                IF (configuration.power.syncMotionSimulation = TRUE) THEN
                   (* SynchroniziedMotionSimulation is set*)
                    IF (tempEnableAxis = FALSE) AND (statEnableAxisOld = TRUE) THEN
                       (* Falling edge at enableAxis --> set simulation*)
                        statSyncMotionSimulationState := AXIS_STATE_SET_SIM;
                        statEnableAxis                := TRUE;
                        tempStateChangeActive         := TRUE;
                    ELSE
                       (* FALSE or rising edge at input enableAxis*)
                        statEnableAxis := tempEnableAxis;
                    END_IF;

                ELSE
                   (* SynchroniziedMotionSimulation not set*)
                   (* MC_POWER is only controlled by enableAxis input*)
                    statEnableAxis := tempEnableAxis;
                END_IF;

            AXIS_STATE_SET_SIM:
				(*
                (* Set the axis in simulation*)
                (*----------------------------------------------------------*)
                (* Enable SynchronizedMotionSimulation*)
				*)
                instSyncMotionSimulation(Slave := axis,
                                         Enable := TRUE);
				(*
                (*----------------------------------------------------------*)
				*)
				
                IF (instSyncMotionSimulation.InSimulation = TRUE) THEN
                    statEnableAxis := FALSE;
                   (* Axis in Simulation - Change state*)
                    statSyncMotionSimulationState := AXIS_DISABLE;

                ELSIF (instSyncMotionSimulation.Error = TRUE) THEN
                   (* Error occurred - Disable Axis immediately*)
                    statEnableAxis                := FALSE;
                    statSyncMotionSimulationState := AXIS_STATE_RESET_SIM;

                ELSE
                    ;(* Wait for Axis is in simulation*)
                END_IF;

            AXIS_DISABLE:

                (* Disable axis*)
                (*----------------------------------------------------------*)
                (* Enable SynchronizedMotionSimulation*)

                instSyncMotionSimulation(Slave := axis,
                                         Enable := TRUE);

                (*----------------------------------------------------------*)


                IF (instPower.Error = TRUE) THEN
                    statSyncMotionSimulationState := AXIS_STATE_RESET_SIM;
                ELSIF (instPower.Status = FALSE) THEN
                   (* Axis disabled*)
                    statSyncMotionSimulationState := AXIS_STATE_IN_SIM;
                ELSE
                    ;(* Wait for Axis is disabled*)
                END_IF;

            AXIS_STATE_IN_SIM:

                (* Axis is in simulation*)
                (*----------------------------------------------------------*)
                (* Enable SynchronizedMotionSimulation*)

                instSyncMotionSimulation(Slave := axis,
                                         Enable := TRUE);

                (*----------------------------------------------------------*)

				
                IF (tempEnableAxis = TRUE) AND (statEnableAxisOld = FALSE) THEN
                   (* Rising edge at enableAxis --> reset simulation*)
                    statSyncMotionSimulationState := AXIS_ENABLE;
                    statEnableAxis                := TRUE;
                    tempStateChangeActive         := TRUE;
                ELSIF (configuration.power.syncMotionSimulation = FALSE) THEN
                   (* End of synchronizedMotionSimulation by configuration without starting Axis*)
                    statSyncMotionSimulationState := AXIS_STATE_RESET_SIM;
                    tempStateChangeActive         := TRUE;

                ELSE
                    ;(* Wait for rising egde at enableAxis*)
                END_IF;

            AXIS_ENABLE:

                (* Enable Axis*)
                (*----------------------------------------------------------*)
                (* Enable SynchronizedMotionSimulation while axis is enabling*)
				
                instSyncMotionSimulation(Slave := axis,
                                         Enable := TRUE);


                (*----------------------------------------------------------*)
                (* Read Statusword only when not already read out*)

                IF (tempStatusWord = 16#0)
                    THEN

                    (*tempStatusWord :=  axis.StatusWord;*)
                    tempStatusWord := axis.NcToPlc.StateDWord;

                END_IF;

                IF (tempEnableAxis = FALSE) AND (statEnableAxisOld = TRUE) THEN
                    statSyncMotionSimulationState := AXIS_STATE_RESET_SIM;
                    statEnableAxis                := FALSE;

                ELSIF (tempStatusWord.0 = TRUE) OR (instPower.Error = TRUE)
               (* Reset simulation if axis is enabled or MC_POWER.STATUS = FALSE (Axis Error)*)
                    THEN
                   (* FALSE on enable input*)
                    statSyncMotionSimulationState := AXIS_STATE_RESET_SIM;
                    tempStateChangeActive         := TRUE;

                ELSE
                    ;(* Wait for Axis is Enabled*)
                END_IF;

            AXIS_STATE_RESET_SIM:

                (* Reset the axis simulation*)
                (*----------------------------------------------------------*)
                (*Enable SynchronizedMotionSimulation*)
				

                instSyncMotionSimulation(Slave := axis,
                                         Enable := FALSE);

                (*----------------------------------------------------------*)

				
                IF (instSyncMotionSimulation.InSimulation = FALSE) AND
                    (instSyncMotionSimulation.Busy = FALSE)
                    THEN
                   (* Axis simulation is disabled*)
                    statSyncMotionSimulationState := AXIS_NOT_IN_SIM;

                ELSE
                    ;(* Wait for axis simulation is disabled*)
                END_IF;

                IF (tempEnableAxis = FALSE) AND (statEnableAxisOld = TRUE) THEN
                    statEnableAxis := FALSE;
                END_IF;

        ELSE
           (* Errorhandling*)
            statStatus                          := ERR_UNDEFINED_MOTION_SIMULATION_STATE;
            statErrorUserCleared                := TRUE;
            diagnostics.subfunctionStatus       := 0;
            diagnostics.basicMotionState        := statBasicMotionState;
            diagnostics.superimposedMotionState := statSupImpMotionState;
           (* Set error state*)
            statFBState := FB_ERROR;
        END_CASE;
    UNTIL (tempStateChangeActive = FALSE)
    END_REPEAT;

   (* Evaluation of MC_Command*)
    IF (instSyncMotionSimulation.Error = TRUE) AND (statSynchronizedMotionErrorOld = FALSE) THEN
       (* Errorhandling - Set error only at rising edge*)
        statErrorAutoCleared                := TRUE;
        statStatus                          := ERR_MC_SYNCHRONIZEDMOTIONSIMULATION;
        diagnostics.basicMotionState        := statBasicMotionState;
        diagnostics.superimposedMotionState := statSupImpMotionState;
        diagnostics.subfunctionStatus       := instSyncMotionSimulation.ErrorId;

    ELSIF (instSyncMotionSimulation.Error = FALSE) AND (statStatus = ERR_MC_SYNCHRONIZEDMOTIONSIMULATION)
        THEN
       (* Reset error if error gone at respective Status*)
        statErrorAutoCleared := FALSE;
        statStatus           := STATUS_SUBSEQUENT_CALL;
    ELSE
        ;
    END_IF;

    statSynchronizedMotionErrorOld := instSyncMotionSimulation.Error;
    tempEnableAxis                 := statEnableAxis;
    {END_REGION}

   (* Enable and disable axis*)
    {REGION "POWER"}
   (* Call MC_POWER*)
    instPower(Axis := axis,
              	Enable := tempEnableAxis,
              	Enable_Positive := TRUE,
            	Enable_Negative := TRUE,
    		(*StartMode :=  configuration.power.startMode,
	         StopMode :=  configuration.power.stopMode*) );

   (* Set and Reset of Error*)
    IF (instPower.Error = TRUE) AND
        ((statStatus = STATUS_SUBSEQUENT_CALL) OR (statPowerErrorOld = FALSE))
        THEN
       (* Error is set at rising edge of MC_POWER.Error*)
       (* Errorhandling*)
        statStatus                              := ERR_MC_POWER;
        statErrorAutoCleared                    := TRUE;
        statDiagnostics.basicMotionState        := statBasicMotionState;
        statDiagnostics.superimposedMotionState := statSupImpMotionState;
        statDiagnostics.subfunctionStatus       := instPower.ErrorId;
        diagnostics                             := statDiagnostics;

    ELSIF (statStatus = ERR_MC_POWER) AND (instPower.Error = FALSE)
        THEN
       (* Reset Error*)
        statStatus           := STATUS_SUBSEQUENT_CALL;
        statErrorAutoCleared := FALSE;

    ELSIF (tempEnableAxis = TRUE) AND (statEnableAxisOld = FALSE) THEN
       (* Reset Error*)
        statStatus           := STATUS_SUBSEQUENT_CALL;
        statErrorAutoCleared := FALSE;
        diagnostics          := statEmptyDiagnostics;
        statDiagnostics      := statEmptyDiagnostics;

    ELSE
        ;(* Do nothing*)
    END_IF;
    {END_REGION}
    {END_REGION}
END_IF;

{END_REGION}


(*----------------------------------------------------------------------------------------------*)
(*FB Statemachine *)
(*----------------------------------------------------------------------------------------------*)


{REGION "FB_STATEMACHINE"}
CASE statFBState OF
    AXIS_MOTION:
       (* Check command inputs*)
        IF (statExtendedCommand = CMD_NO_SELECTION) AND (statBasicCommand = CMD_NO_SELECTION) AND (statSupImpCommand = CMD_NO_SELECTION)
            THEN
           (* Command is reset*)
            IF (instPower.Error = TRUE) THEN
               (* Errorhandling*)
                statStatus           := ERR_MC_POWER;
                statErrorAutoCleared := TRUE;
                diagnostics          := statDiagnostics;
            ELSIF (instSyncMotionSimulation.Error = TRUE) THEN
                ;(* Do nothing*)

            ELSIF (instTorqueLimiting.Error = TRUE) THEN
                ;(* Do nothing. V1.00.03 dont reset IF torque limiting  error is pending *)

            ELSE
               (* Reset Error only if no Error at MC_POWER is present*)
                statStatus           := STATUS_SUBSEQUENT_CALL;
                statErrorAutoCleared := FALSE;
            END_IF;

        ELSIF (statExtendedCommand = statExtendedCommandOld) AND
            (statBasicCommand = statBasicCommandOld) AND
            (statSupImpCommand = statSupImpCommandOld)
            THEN
            ;(* No change at command - do nothing*)

        ELSE
           (* Command changed*)
            tempNewExtendedCmd    := NO_SELECTION;
            tempNewBasicMotionCmd := NO_SELECTION;
            tempNewSupImpCmd      := NO_SELECTION;
            tempErrorInCmd        := FALSE;

            {REGION "CHECK BASIC_MOTION_CMD"}
           (* Check basic motion command*)
            IF (statBasicCommand = statBasicCommandOld) THEN
                ;(* Do nothing*)
            ELSE
               (* Evaluate rising edges for basic motion command word - all rising edges of basic command word saved in tempRisingBasicCmd*)
                tempRisingCmd     := ((statBasicCommand XOR statBasicCommandOld) AND statBasicCommand);
                tempCountRisEdges := 0;(* Initialize counter for rising edges*)
               (* Count rising edges in tempRisingBasicCmd*)
                FOR tempIndex := BITPOSITION_BASIC_MOTION_CMD TO BIT_POS_LAST DO
                    tempDword := SHR(tempRisingCmd, INT_TO_USINT(tempIndex));
                   (* Check for rising edge*)
                    IF (tempDword.0 = TRUE) THEN
                        tempCountRisEdges := tempCountRisEdges + 1;(* Increment at rising edge*)
                    END_IF;
                END_FOR;

                IF (tempRisingCmd.2 = TRUE) OR (tempRisingCmd.3 = TRUE) THEN
                    tempCountRisEdges := tempCountRisEdges + 1;(* jogForward AND/OR jogBackward is standing for 1 Command/rising edge*)
                END_IF;

               (* Check Basic motion command*)
                IF (tempCountRisEdges = 1) OR
                    (tempRisingCmd.0 = TRUE)(* fastStop selected*)
                    OR
                    (tempRisingCmd.1 = TRUE)(* Stop selected*)
                    THEN
                   (* Valid basic motion command selected*)
                    IF (tempRisingCmd.0 = TRUE)
                        THEN
                       (* FastStop selected*)
                        statFBState           := AXIS_FAST_STOPPING;
                        tempNewBasicMotionCmd := FAST_STOP_SELECTED;
                        tempStopCmdSelected   := TRUE;
                    ELSIF (tempRisingCmd.1 = TRUE)
                        THEN
                       (* Stop selected*)
                        tempNewBasicMotionCmd := STOP_SELECTED;
                        tempStopCmdSelected   := TRUE;
                    ELSE
                       (* Valid basic command priority 3 selected*)
                       (* Set basic motion state*)
                        tempNewBasicMotionCmd := DWORD_TO_DINT(tempRisingCmd);
                    END_IF;

                ELSIF (tempCountRisEdges > 1) THEN
                   (* Errorhandling - Invalid command *)
                    statStatus     := ERR_INVALID_BASIC_MOTION_CMD;
                    tempErrorInCmd := TRUE;

                ELSE
                    ;(* Falling edge detection*)
                END_IF;
            END_IF;

            {END_REGION}
            {REGION "CHECK_SUP_IMP_CMD"}
           (* Check superimposed motion command*)
            IF (statSupImpCommand = statSupImpCommandOld) THEN
                ;(* Do nothing*)
            ELSE
               (* Superimposed motion command selected *) 
                IF (tempErrorInCmd = FALSE) AND(* No Stop command selected in current cycle*)
                    (tempStopCmdSelected = FALSE)
                    THEN
                    tempRisingCmd     := ((statSupImpCommand XOR statSupImpCommandOld) AND statSupImpCommand);
                    tempCountRisEdges := 0;(* Initialize counter for rising edges*)
                   (* Count rising edges in tempRisingSupImpCmd*)
                    FOR tempIndex := BITPOSITION_SUPERIMPOSED_MOTION_CMD TO BIT_POS_LAST DO
                        tempDword := SHR(tempRisingCmd, INT_TO_USINT(tempIndex));
                       (* Check for rising edge*)
                        IF (tempDword.0 = TRUE) THEN
                            tempCountRisEdges := tempCountRisEdges + 1;
                        END_IF;
                    END_FOR;

                    IF (tempCountRisEdges = 1) THEN
                       (* Valid superimposed motion command*)
                        tempNewSupImpCmd := DWORD_TO_DINT(tempRisingCmd);

                    ELSIF (tempCountRisEdges > 1) THEN
                       (* Invalid Superimposed motion command*)
                        statStatus     := ERR_INVALID_SUPERIMPOSED_MOTION_CMD;
                        tempErrorInCmd := TRUE;

                    ELSE
                        ;(* Falling edge detection*)
                    END_IF;

                ELSE
                    ;(* Stop or Faststop command selected OR error in BasicCommand*)
                END_IF;
            END_IF;

            {END_REGION}
            {REGION "CHECK_EXT_CMD"}
           (* Check extended command (reset, homing, torquelimiting)*)
            IF (statExtendedCommand = statExtendedCommandOld) THEN
                ;(* Do nothing*)
            ELSE
               (* Extended command selected*)
                IF (tempErrorInCmd = FALSE)
                    THEN
                    tempRisingCmd := ((statExtendedCommand XOR statExtendedCommandOld) AND statExtendedCommand);
                   (* Rising edge on torquelimiting command*)
                    IF (tempRisingCmd.1 = TRUE)
                        THEN
                        tempNewExtendedCmd.1 := TRUE;
                       (* Rising Edge at Homing on Fixed Stop and Torquelimiting*)
                        IF (tempNewBasicMotionCmd.10 = TRUE) AND (configuration.homing.extendedMode = 0) THEN
                            ;(* Errorhandling*)
                            statStatus           := ERR_INVALID_EXTENDED_CMD;
                            tempErrorInCmd       := TRUE;
                            tempNewExtendedCmd.1 := FALSE;

                           (* Check if torquelimiting is not for use in homing on fixed stop function*)
                        ELSIF (statTorqueLimitingState = TORQUE_LIMTING_SELECTED)
                       (* OR ( statTorqueLimitingState =  AUTOMATIC_MODE_CHANGE) V1.00.03 Not required anymore*)
                            THEN
                            ;(* Torquelimiting already busy no need of restart*)
                           (* tempNewExtendedCmd.1 := FALSE; // V1.0.4 Initialize Diagnostics at rising edge of torquelimiting*)

                        ELSIF (statTorqueLimitingState = FIXED_STOP_DETECTION_ACTIVE)
                            THEN
                            ;(* Torquelimiting rejected because MC_Torquelimiting is used during homing on fixed stop functionality*)
                            statStatus           := ERR_TORQUE_LIMITING_NOT_ALLOWED;
                            tempErrorInCmd       := TRUE;
                            tempNewExtendedCmd.1 := FALSE;

                        ELSE
                            ;(* Start torquelimiting functionality*)
                        END_IF;
                    END_IF;

                   (* Rising edge on passive homing command*)
                    IF (tempRisingCmd.2 = TRUE)
                        THEN
                        tempNewExtendedCmd.2 := TRUE;
                        IF (statBasicMotionState = ACTIVE_HOMING_SELECTED) AND
                            (statActiveHomingState = HOMING_ON_FIXED_STOP) AND
                            (statExeOfBasicMotion = CMD_BUSY)
                            THEN
                           (* Passive Homing selected at homing on fixed stop *)
                            statStatus           := ERR_HOMING_MODE_NOT_ALLOWED;
                            tempErrorInCmd       := TRUE;
                            tempNewExtendedCmd.2 := FALSE;
                        ELSE
                            ;(* No error occurred*)
                        END_IF;
                    END_IF;
                ELSE
                    ;(* Error in basic motion command or superimposed motion command *)
                END_IF;
            END_IF;

            {END_REGION}
           (* Enable commands*)
            IF (tempErrorInCmd = TRUE) AND (tempStopCmdSelected = FALSE)
                THEN
               (* Error in current command - No Execution*)
                statErrorAutoCleared          := TRUE;
                diagnostics.subfunctionStatus := 0;
               (* Write diagnostics*)
                statDiagnostics.basicMotionState        := statBasicMotionState;
                statDiagnostics.superimposedMotionState := statSupImpMotionState;
                statResetIncJog                         := TRUE;
               (* Set next state*)
                statFBState := AXIS_STOP_ON_ERROR_SELECTION;
            ELSE
               (* No Error in command occurred*)
                IF (
                    (tempNewExtendedCmd <> NO_SELECTION) OR (tempNewBasicMotionCmd <> NO_SELECTION) OR (tempNewSupImpCmd <> NO_SELECTION)
                    ) OR
                    (tempStopCmdSelected = TRUE)
                    THEN
                    {REGION "ENABLE_BASIC_MOTION_CMD"}
                   (* New valid command selected*)
                   (* Basic motion commands*)
                    IF (tempNewBasicMotionCmd <> NO_SELECTION) THEN
                       (* Reset of waiting Gearin / camIn command*)
                        IF (configuration.generalSettings.abortWaitingSyncCmd = TRUE) AND
                            (((statBasicMotionState = GEAR_IN_ABSOLUTE_SELECTED) AND (statExeOfBasicMotion = CMD_BUSY))(* GearInAbsolute waiting*)
                            OR
                            ((statBasicMotionState = CAM_IN_SELECTED) AND (statExeOfBasicMotion = CMD_BUSY)))(* CamIn waiting*)
                            THEN
                            statMainSelectionState := RESET_GEARING;(* Reset waiting absolute gearing / camIn command *)
                            instGearIn(Master := master,
                                       Slave := axis,
                                       Execute := FALSE);
                        ELSE
                            statMainSelectionState := CALL_BASIC_MOTION;
                        END_IF;

                        statFirstCycleBasicMotion := TRUE;
                       (* Evaluate if Jog command is set*)
                        IF (tempNewBasicMotionCmd.2 = TRUE) OR (tempNewBasicMotionCmd.3 = TRUE)
                            THEN
                            statExeOfBasicMotion := CMD_BUSY;
                           (* Select Jogmode*)
                            IF ((statBasicCommand.2 = FALSE) AND (tempNewBasicMotionCmd.3 = TRUE)
                                ) OR(* Rising edge at JogBackward and JogForward = FALSE*)
                                ((statBasicCommand.3 = FALSE) AND (tempNewBasicMotionCmd.2 = TRUE)
                                ) OR(* Only rising edge at JogForward and Jogbackward = FALSE*)
                                ((tempNewBasicMotionCmd.2 = TRUE) AND (tempNewBasicMotionCmd.3 = TRUE)
                                )(* Rising edge at FW and BW*)
                                THEN
                               (* One Input direction = False, other is rising edge, or both rising edge --> Start jog*)
                                IF (statJogMode <> configuration.jog.mode) THEN
                                    statResetIncJog := TRUE;
                                END_IF;

                                statJogMode := configuration.jog.mode;
                            ELSE
                                ;(* Rising edge at one input, the other is already TRUE - Dont Change Jogmode*)
                                IF ((statBasicMotionState = JOG_BACKWARD_SELECTED) OR (statBasicMotionState = JOG_FORWARD_SELECTED)) AND
                                    (statJogMode <> JOG_MODE_CONTINUOUS)
                                    THEN
                                    statFirstCycleBasicMotion := FALSE;
                                END_IF;
                            END_IF;

                        ELSE
                            ;(* Reset jog increment if other command than jog selected*)
                            statResetIncJog := TRUE;
                        END_IF;

                       (* Set new basic motion state*)
                        statBasicMotionState := tempNewBasicMotionCmd;
                    END_IF;

                    {END_REGION}
                    {REGION "ENABLE_SUP_IMP_CMD"}
                   (* Superimposed motion commands*)
                    IF (tempNewSupImpCmd <> NO_SELECTION) THEN
                        statSupImpMotionState      := tempNewSupImpCmd;
                        statFirstCycleSupImpMotion := TRUE;
                        statResetIncJog            := TRUE;
                    END_IF;

                    {END_REGION}
                   (* Extended commands*)
                    {REGION "ENABLE_EXT_CMD"}
                    IF (tempNewExtendedCmd <> NO_SELECTION) THEN
                        IF (tempNewExtendedCmd.1 = TRUE) THEN
                           (* Rising edge on torquelimiting command*)
                            IF (statTorqueLimitingState = NO_TORQUE_LIMITING_ACTIVE)
                                THEN
                               (* No torquelimiting active --> Enable torquelimiting*)
                                statTorqueLimitingState := TORQUE_LIMTING_SELECTED;
                            ELSE
                                ;(* Torquelimiting already active*)
                               (* statTorqueLimitingState :=  AUTOMATIC_MODE_CHANGE; V1.00.03 Not required anymore *)
                            END_IF;
                        END_IF;

                       (* Homing command*)
                        IF (tempNewExtendedCmd.2 = TRUE) THEN
                            statPassiveHomingState := configuration.homing.extendedMode;
                            statFirstCycleHoming   := TRUE;
                            statResetIncJog        := TRUE;
                        END_IF;
                    END_IF;

                    {END_REGION}
                   (* Reset error*)
                    statStatus           := STATUS_SUBSEQUENT_CALL;
                    statErrorAutoCleared := FALSE;
                    diagnostics          := statEmptyDiagnostics;
                    statDiagnostics      := statEmptyDiagnostics;

                ELSE
                    ;(* No rising edge at commands*)
                END_IF;
            END_IF;
        END_IF;

    AXIS_FAST_STOPPING:
        IF (configuration.fastStop.replaceStopPossible = FALSE) THEN
            ;(* Fast stop command can not be interrupted by another command*)
           (* State change is executed in FastStop implementation if command finished *)
        ELSE
            statFBState := AXIS_MOTION;
        END_IF;

    AXIS_STOP_ON_ERROR_SELECTION,
        AXIS_STOP_ON_ERROR_EXECUTION:
        ;    (* Wait for stopping axis if StopOnError is configured*)
    FB_ERROR:(* Error state*)
        ;    (* Do nothing, status already set*)

ELSE
   (* Errorhandling*)
    statStatus                          := ERR_UNDEFINED_FB_STATE;
    statErrorUserCleared                := TRUE;
    diagnostics.subfunctionStatus       := 0;
    diagnostics.basicMotionState        := statBasicMotionState;
    diagnostics.superimposedMotionState := statSupImpMotionState;
   (* Set error state*)
    statFBState := FB_ERROR;
END_CASE;

{END_REGION}


(*----------------------------------------------------------------------------------------------*)
(*Execution of reset functionality*)
(*----------------------------------------------------------------------------------------------*)


{REGION "EXECUTION_OF_RESET_COMMAND"}
(* Firstcycle of command*)

IF (statExtendedCommand.0 = TRUE) AND (statExtendedCommandOld.0 = FALSE) THEN
    statFirstCycleReset := TRUE;
   (* Reset MC_RESET command*)
    instReset(Axis := axis,
              Execute := FALSE);

    statFirstCycleResetError := FALSE;
    statResetState           := CMD_BUSY;
END_IF;

CASE statResetState OF
    CMD_IDLE:
        ;(* Do nothing*)

    CMD_BUSY:
       (* Call MC_Command*)
        instReset(Axis := axis,
                  Execute := statExtendedCommand.0,
        (*Restart :=  configuration.generalSettings.resetWithRestart*) );

       (* Evaluate MC_Command*)
        IF (instReset.Error = TRUE) THEN
           (* Errorhandling*)
            IF (statFirstCycleResetError = FALSE) THEN
                statErrorAutoCleared                := TRUE;
                diagnostics.status                  := ERR_MC_RESET;
                statStatus                          := ERR_MC_RESET;
                diagnostics.basicMotionState        := statBasicMotionState;
                diagnostics.superimposedMotionState := statSupImpMotionState;
                diagnostics.subfunctionStatus       := instReset.ErrorId;
                statFirstCycleResetError            := TRUE;
               (* Set next state*)
                statResetState := CMD_IDLE;
                IF (statFBState = AXIS_MOTION) THEN
                   (* Set TO_STOP_ON_ERROR State only if the current state is TO_MOTION*)
                    statFBState := AXIS_STOP_ON_ERROR_SELECTION;
                END_IF;
            END_IF;

        ELSIF (instReset.Busy = FALSE) THEN
           (* Set next state*)
            statResetState := CMD_IDLE;
        ELSE
            ;(* Command selected*)
        END_IF;

ELSE
   (* Errorhandling  *)  
    statStatus                              := ERR_UNDEFINED_RESET_STATE;
    statErrorUserCleared                    := TRUE;
    diagnostics                             := statDiagnostics;
    diagnostics.subfunctionStatus           := 0;
    statDiagnostics.basicMotionState        := statBasicMotionState;
    statDiagnostics.superimposedMotionState := statSupImpMotionState;
END_CASE;

{END_REGION}


(*----------------------------------------------------------------------------------------------*)
(* Execution of functionalities of basic coordinate system*)
(*----------------------------------------------------------------------------------------------*)


{REGION "EXECUTION_OF_BASIC_MOTION_COMMANDS"}
(*Statemachine for basic motion commands*)

(*Write diagnostics*)
statDiagnostics.basicMotionState        := statBasicMotionState;
statDiagnostics.superimposedMotionState := statSupImpMotionState;
REPEAT
    tempStateChangeActive := FALSE;
   (* Statemachine for main selection state*)
    CASE statMainSelectionState OF
        CALL_BASIC_MOTION:
            CASE statBasicMotionState OF
                NO_SELECTION:
                    ;(* No execution*)

                FAST_STOP_SELECTED:
                    ;(* Implementation at end of code*)

                STOP_SELECTED:
                   (* No additional features*)
                    {REGION "STOP_SELECTED"}
                   (* Firstcycle of command*)
                    IF (statFirstCycleBasicMotion = TRUE) THEN
                       (* Reset HALT command*)
                        instHalt(Axis := axis,
                                 Execute := FALSE);
                    END_IF;

                   (* Call MC_Command*)
                    instHalt(Axis := axis,
                             Execute := statBasicCommand.1 OR statFirstCycleBasicMotion,
                             Deceleration := configuration.stop.deceleration,
                             (*AbortAcceleration :=  configuration.stop.abortAcceleration,*)
                             Jerk := configuration.stop.jerk);

                   (* Evaluate MC_Command*)
                    IF (instHalt.Busy = FALSE) AND
                        (instHalt.Error = FALSE) AND
                        (instHalt.Done = FALSE) AND
                        (instHalt.CommandAborted = FALSE)
                        THEN
                       (* Return to NO_SELECTION if command finished*)
                        statBasicMotionState := NO_SELECTION;

                    ELSIF (instHalt.Error = TRUE)
                        THEN
                       (* Errorhandling*)
                        statStatus                    := ERR_MC_HALT;
                        statErrorAutoCleared          := TRUE;
                        diagnostics                   := statDiagnostics;
                        diagnostics.subfunctionStatus := instHalt.ErrorId;
                       (* Set next state*)
                        statFBState          := AXIS_STOP_ON_ERROR_SELECTION;
                        statBasicMotionState := NO_SELECTION;
                    ELSE
                        ;(* Command selected*)
                    END_IF;

                   (* Write MC_Command outputs to internal variable*)
                    statExeOfBasicMotion   := 16#0;
                    statExeOfBasicMotion.0 := instHalt.Busy;
                    statExeOfBasicMotion.1 := instHalt.Done;
                    statExeOfBasicMotion.2 := instHalt.CommandAborted;
                    statExeOfBasicMotion.3 := instHalt.Error;
                {END_REGION}

                JOG_FORWARD_SELECTED, JOG_BACKWARD_SELECTED, JOG_FW_AND_BW_SELECTED:
                   (* Additional features (applicative): Jog mode incremental*)
                    {REGION "JOG_SELECTED"}
                    CASE statJogMode OF
                        JOG_MODE_CONTINUOUS:
                            {REGION "JOG_MODE_CONTINUOUS"}
                           (* No additional feature*)
                           (* Firstcycle of command*)
                            IF (statFirstCycleBasicMotion = TRUE) THEN
                               (* No of dynmics into static variables because changes are accepted by MC_JOG immetiately (enable)*)
                                instMoveJog(Axis := axis,
                                            JogForward := FALSE,
                                            JogBackwards := FALSE);
                            END_IF;

                           (* Call MC_Command*)
                            instMoveJog(Axis := axis,
                                        JogForward := statBasicCommand.2,
                                        JogBackwards := statBasicCommand.3,
                                        Velocity := configuration.jog.velocity,
                                        Acceleration := configuration.jog.acceleration,
                                        Deceleration := configuration.jog.deceleration,
                                        (*PositionControlled :=  configuration.jog.positionControlled,*)
				Mode := 2,
                                        Jerk := configuration.jog.jerk);

                           (* Evaluate MC_Command*)
                            IF (instMoveJog.Busy = FALSE) AND
                                (instMoveJog.Error = FALSE) AND
                                (instMoveJog.CommandAborted = FALSE) (*AND
	                      ( instMoveJog.InVelocity = FALSE)*)
                                THEN
                               (* Return to NO_SELECTION if command finished*)
                                statBasicMotionState := NO_SELECTION;

                            ELSIF (instMoveJog.Error = TRUE)
                                THEN
                               (* Errorhandling*)
                                statStatus                    := ERR_MC_MOVEJOG;
                                statErrorAutoCleared          := TRUE;
                                diagnostics                   := statDiagnostics;
                                diagnostics.subfunctionStatus := instMoveJog.ErrorId;
                               (* Set next state*)
                                statBasicMotionState := NO_SELECTION;
                                statFBState          := AXIS_STOP_ON_ERROR_SELECTION;

                            ELSE
                                ;(* Command selected*)
                            END_IF;

                           (* Write MC_Command outputs to internal variable*)
                            statExeOfBasicMotion   := 16#0;
                            statExeOfBasicMotion.0 := instMoveJog.Busy;
                            statExeOfBasicMotion.2 := instMoveJog.CommandAborted;
                            statExeOfBasicMotion.3 := instMoveJog.Error;
                            (*statExeOfBasicMotion.4 := instAxisStatus.stAxisStatus.ConstantVelocity; (*####*)*)
				  statExeOfBasicMotion.4 := axis.Status.ConstantVelocity;
                        {END_REGION}

                        JOG_MODE_CONTINUE_INCREMENT, JOG_MODE_NEW_INCREMENT:
                            {REGION "JOG_MODE_INCREMENTAL"}
                           (* This case is additional feature (MC_MOVERELATIVE and MC_HALT internal used)*)
                            CASE statExeOfBasicMotion OF
                                CMD_BUSY:
                                   (* Firstcycle of command*)
                                    IF (statFirstCycleBasicMotion = TRUE) THEN(*New rising edge at JogForward or JogBackard*)
                                       (* Check for only one Jog direction selected (Forward OR Backward)*)
                                        IF (statBasicCommand.2 XOR statBasicCommand.3)(* Only one direction selected*)
                                            THEN
                                           (* Reset MOVERELATIVE command*)
                                            instMoveRelative(Axis := axis,
                                                             Execute := FALSE);

                                           (* Reset HALT command*)
                                            instHalt(Axis := axis,
                                                     Execute := FALSE);

                                           (* Set new Increment if direction changed neccesary*)
                                            IF (statResetIncJog = FALSE) THEN
                                                IF ((statIncJogDirectionOld = FORWARD_DIR) AND (statBasicCommand.2 = TRUE)) OR
                                                    ((statIncJogDirectionOld = BACKWARD_DIR) AND (statBasicCommand.3 = TRUE))
                                                    THEN
                                                    ;(* Direction of last jog process same as current --> continue Jog*)
                                                ELSE
                                                    statResetIncJog := TRUE;
                                                END_IF;
                                            END_IF;

                                           (* Determine distance for positioning command (relative)*)
                                            IF (configuration.jog.mode = JOG_MODE_NEW_INCREMENT)(* In this mode a new increment is always set*)
                                                OR
                                                ((configuration.jog.mode = JOG_MODE_CONTINUE_INCREMENT) AND (statResetIncJog = TRUE))
                                                THEN
                                                statResetIncJog := FALSE;
                                               (* New increment*)
                                                (*statIncJogStartPosition :=  axis.Position;*)              (* Targetposition for increment*)
                                                statIncJogStartPosition := axis.NcToPlc.ActPos;             (* Targetposition for increment*)
                                                statIncrement           := ABS(configuration.jog.increment);(* absolut Distance for increment*)
                                                IF (statBasicCommand.2 = TRUE) THEN
                                                   (* JogForward selected*)
                                                    statPosition           := ABS(configuration.jog.increment);
                                                    statIncrement          := statPosition;
                                                    statIncJogDirectionOld := FORWARD_DIR;
                                                ELSIF (statBasicCommand.3 = TRUE) THEN
                                                   (* JogBackward selected*)
                                                    statPosition           := -ABS(configuration.jog.increment);
                                                    statIncrement          := statPosition;
                                                    statIncJogDirectionOld := BACKWARD_DIR;
                                                ELSE
                                                   (* Normal not possible to reach ELSE-branch*)
                                                    statIncJogDirectionOld := 0;
                                                END_IF;

                                            ELSE
                                               (* Check for modulo axis*)
                                                (*IF ( axis.Modulo.Enable = FALSE) THEN*)
                                                IF (tempFalse = TRUE) THEN
                                                   (* No Modulo enabled*)
                                                   (* Continue increment*)

                                                    statPosition := (statIncJogStartPosition + statIncrement) - axis.NcToPlc.ActPos;
                                                   (* Distance   :=            setpoint                         - actualvalue*)
                                                ELSE
                                                   (* Modulo enabled*)
                                                    statPosition := statIncJogDistance;
                                                END_IF;

                                            END_IF;

                                            statIncJogSubState := INC_JOG_START;

                                           (* Store Dynamics*)
                                            statVelocity     := ABS(configuration.jog.velocity);
                                            statAcceleration := configuration.jog.acceleration;
                                            statDeceleration := configuration.jog.deceleration;
                                            statJerk         := configuration.jog.jerk;

                                        ELSE
                                           (* Errorhandling - Invalid direction (forward and backward selected)*)
                                            statStatus                    := ERR_INVALID_JOG_DIR;
                                            statErrorAutoCleared          := TRUE;
                                            diagnostics.subfunctionStatus := 0;
                                            diagnostics.basicMotionState  := statBasicMotionState;
                                           (* Set next state*)
                                            statFBState          := AXIS_STOP_ON_ERROR_SELECTION;
                                            statBasicMotionState := NO_SELECTION;
                                            statExeOfBasicMotion := CMD_ERROR;
                                            statIncJogSubState   := INC_JOG_IDLE;
                                        END_IF;

                                    ELSIF ((statBasicCommand.2 = FALSE) AND (statBasicCommand.3 = FALSE))(* No jog input selected --> Stop moving*)
                                        AND
                                        (statIncJogSubState <> INC_JOG_STOP)
                                        THEN
                                       (* Reset HALT command*)
                                        instHalt(Axis := axis,
                                                 Execute := FALSE);

                                        statIncJogSubState := INC_JOG_STOP;
                                        (*statIncJogDistance :=  axis.StatusPositioning.Distance;*)

                                    ELSIF (statBasicCommand.2 = TRUE) AND (statBasicCommand.3 = TRUE)(* jogForward and jogBackward selected - Error*)
                                        THEN
                                       (* Reset HALT command*)
                                        instHalt(Axis := axis,
                                                 Execute := FALSE);

                                        statIncJogSubState := INC_JOG_STOP;
                                       (* Errorhandling*)
                                        statStatus                    := ERR_INVALID_JOG_DIR;
                                        statErrorAutoCleared          := TRUE;
                                        diagnostics                   := statDiagnostics;
                                        diagnostics.subfunctionStatus := 0;
                                       (* Set next state*)
                                        statExeOfBasicMotion := CMD_ERROR;
                                        statBasicMotionState := NO_SELECTION;
                                        statFBState          := AXIS_STOP_ON_ERROR_SELECTION;
                                    ELSE
                                        ;(* Command running*)
                                    END_IF;

                                   (* Select motion*)
                                    CASE statIncJogSubState OF
                                        INC_JOG_IDLE:
                                            ;(* Do nothing - Error occurred (jogforward and jogbackward are set in firstCycle of operation)*)

                                        INC_JOG_START:(* Run jog operation --> Motion stops automatically if increment complete*)
                                            instMoveRelative(Axis := axis,
                                                             Execute := TRUE,
                                                             Distance := statPosition,
                                                             Velocity := statVelocity,
                                                             Acceleration := statAcceleration,
                                                             Deceleration := statDeceleration,
                                                             Jerk := statJerk);

                                           (* Evaluate MC_Command*)
                                            IF (instMoveRelative.Done = TRUE) THEN
                                               (* Increment completed*)
                                                statResetIncJog := TRUE;
                                               (* Set next state*)
                                                statExeOfBasicMotion := CMD_DONE;
                                                statIncJogSubState   := INC_JOG_IDLE;

                                            ELSIF (instMoveRelative.Error = TRUE) THEN
                                                statResetIncJog := TRUE;
                                               (* Errorhandling*)
                                                statStatus                    := ERR_MC_MOVERELATIVE;
                                                statErrorAutoCleared          := TRUE;
                                                diagnostics                   := statDiagnostics;
                                                diagnostics.subfunctionStatus := instMoveRelative.ErrorId;
                                               (* Set next state*)
                                                statFBState          := AXIS_STOP_ON_ERROR_SELECTION;
                                                statBasicMotionState := NO_SELECTION;
                                                statExeOfBasicMotion := CMD_ERROR;
                                                statIncJogSubState   := INC_JOG_IDLE;

                                            ELSIF (instMoveRelative.CommandAborted = TRUE) THEN
                                                statResetIncJog      := TRUE;
                                                statExeOfBasicMotion := CMD_ABORTED;
                                                statIncJogSubState   := INC_JOG_IDLE;

                                            ELSE
                                               (* statJogDistance :=  axis.StatusPositioning.Distance;*)
                                                ;(* Wait for next state*)
                                            END_IF;

                                        INC_JOG_STOP:(* Executed if inputs are reset --> Stop jog operation OR if jogForward and jogBackward are set --> Error and stop axis*)
                                            instHalt(Axis := axis,
                                                     Execute := TRUE,
                                                     Deceleration := statDeceleration,
                                                     (*AbortAcceleration := FALSE,*)
                                                     Jerk := statJerk);

                                           (* Evaluate MC_Command*)
                                            IF (instHalt.Done = TRUE) THEN
                                               (* Set next state*)
                                                statExeOfBasicMotion := CMD_END_PROCESS;
                                                statIncJogSubState   := INC_JOG_IDLE;

                                            ELSIF (instHalt.Error = TRUE) THEN
                                                statResetIncJog := TRUE;
                                               (* Errorhandling*)
                                                statStatus                    := ERR_MC_HALT;
                                                statErrorAutoCleared          := TRUE;
                                                diagnostics                   := statDiagnostics;
                                                diagnostics.subfunctionStatus := instHalt.ErrorId;
                                               (* Set next state*)
                                                statFBState          := AXIS_STOP_ON_ERROR_SELECTION;
                                                statBasicMotionState := NO_SELECTION;
                                                statExeOfBasicMotion := CMD_ERROR;
                                                statIncJogSubState   := INC_JOG_IDLE;

                                            ELSIF (instHalt.CommandAborted = TRUE) THEN
                                                statResetIncJog := TRUE;
                                               (* Set next state*)
                                                statIncJogSubState   := INC_JOG_IDLE;
                                                statExeOfBasicMotion := CMD_ABORTED;

                                            ELSE
                                                ;(* Wait for stopping axis*)
                                            END_IF;

                                    ELSE
                                       (* Errorhandling*)
                                        statStatus                    := ERR_UNDEFINED_INCREMENTAL_JOG_SUBSTATE;
                                        statErrorUserCleared          := TRUE;
                                        diagnostics                   := statDiagnostics;
                                        diagnostics.subfunctionStatus := 0;
                                       (* Set errorstate*)
                                        statFBState := FB_ERROR;
                                    END_CASE;

                                CMD_DONE,
                                    CMD_ABORTED,
                                    CMD_ERROR,
                                    CMD_END_PROCESS:
                                   (* Return to NO_SELECTION if command finished*)
                                    IF (statBasicCommand.2 = FALSE) AND (statBasicCommand.3 = FALSE)
                                        THEN
                                       (* jogForward and jogbackward inputs are reset*)
                                        statExeOfBasicMotion := CMD_BUSY;
                                        statBasicMotionState := NO_SELECTION;
                                    ELSE
                                        ;(* Wait for falling edge at inputs for jog*)
                                    END_IF;

                            ELSE
                               (* Errorhandling*)
                                statStatus                    := ERR_UNDEFINED_INCREMENTAL_JOG_STATE;
                                statErrorUserCleared          := TRUE;
                                diagnostics.subfunctionStatus := 0;
                                diagnostics.basicMotionState  := statBasicMotionState;
                               (* Set errorstate*)
                                statFBState := FB_ERROR;
                            END_CASE;
                    {END_REGION}

                    ELSE
                       (* Errorhandling - Invalid jog state*)
                        statStatus                    := ERR_INVALID_JOG_MODE;
                        statErrorAutoCleared          := TRUE;
                        diagnostics                   := statDiagnostics;
                        diagnostics.subfunctionStatus := 0;
                       (* Set next state*)
                        statFBState          := AXIS_STOP_ON_ERROR_SELECTION;
                        statBasicMotionState := NO_SELECTION;
                    END_CASE;
                {END_REGION}

                MOVE_VELOCITY_SELECTED:
                   (* Additional features (applicative): Change setpoint on the fly (Velocity) *)
                    {REGION "MOVEVELOCITY_SELECTED"}

                   (* Firstcycle of command*)
                    IF (statFirstCycleBasicMotion = TRUE) THEN
                       (* Reset MC_MOVEVELOCITY command*)
                        instMoveVelocity(Axis := axis,
                                         Execute := FALSE);

                        statVelocityChangeOnTheFly := configuration.moveVelocity.velocityChangeOnTheFly;
                        statVelocity               := configuration.moveVelocity.velocity;          (* Store the last adjusted velocity value*)
                        statAcceleration           := configuration.moveVelocity.acceleration;      (* Store the last adjusted acceleration value*)
                        statDeceleration           := configuration.moveVelocity.deceleration;      (* Store the last adjusted deceleration value*)
                        statJerk                   := configuration.moveVelocity.jerk;              (* Store the last adjusted jerk value*)
                        statDirection              := configuration.moveVelocity.direction;         (* Store the last adjusted axis direction*)
                        statPositionControlled     := configuration.moveVelocity.positionControlled;(* Store the last adjusted motion mode*)

                    ELSIF (statVelocityChangeOnTheFly = TRUE) AND
                        (configuration.moveVelocity.velocity <> statVelocity)(* Velocity changed*)
                        AND
                        (instMoveVelocity.CommandAborted = FALSE)
                        THEN
                       (* Reset MC_MOVEVELOCITY command*)
                        instMoveVelocity(Axis := axis,
                                         Execute := FALSE);

                        statVelocity := configuration.moveVelocity.velocity;(* Store the last adjusted velocity value*)
                    END_IF;

                   (* Call MC_Command*)
                    instMoveVelocity(Axis := axis,
                                     Execute := statBasicCommand.4 OR statFirstCycleBasicMotion,(* Input: moveVelocity*)
                                     Velocity := statVelocity,
                                     Acceleration := statAcceleration,
                                     Deceleration := statDeceleration,
                                     Jerk := statJerk,
                                     Direction := statDirection,
                    (*PositionControlled :=  statPositionControlled,*)
                    (*Current := FALSE*) );

                   (* Evaluate MC_Command*)
                    IF (instMoveVelocity.Busy = FALSE) AND
                        (instMoveVelocity.Error = FALSE) AND
                        (instMoveVelocity.CommandAborted = FALSE) AND
                        (instMoveVelocity.InVelocity = FALSE)
                        THEN
                       (* Return to NO_SELECTION if command finished*)
                        statBasicMotionState := NO_SELECTION;

                    ELSIF (instMoveVelocity.Error = TRUE)
                        THEN
                       (* Errorhandling*)
                        statStatus                    := ERR_MC_MOVEVELOCITY;
                        statErrorAutoCleared          := TRUE;
                        diagnostics                   := statDiagnostics;
                        diagnostics.subfunctionStatus := instMoveVelocity.ErrorId;
                        statVelocityChangeOnTheFly    := FALSE;
                       (* Set next state*)
                        statFBState          := AXIS_STOP_ON_ERROR_SELECTION;
                        statBasicMotionState := NO_SELECTION;

                    ELSE
                        ;(* Command selected*)
                    END_IF;

                   (* Write MC_Command outputs to internal variable*)
                    statExeOfBasicMotion   := 16#0;
                    statExeOfBasicMotion.0 := instMoveVelocity.Busy;
                    statExeOfBasicMotion.2 := instMoveVelocity.CommandAborted;
                    statExeOfBasicMotion.3 := instMoveVelocity.Error;
                    statExeOfBasicMotion.4 := instMoveVelocity.InVelocity;
                {END_REGION}

                POS_RELATIVE_SELECTED:
                   (* Additional features (applicative): Specified direction*)
                    {REGION "POS_RELATIVE_SELECTED"}
                   (* Firstcycle of command*)
                    IF (statFirstCycleBasicMotion = TRUE) THEN
                       (* Configurate the direction of rotation*)
                       (* *)
                        IF ((configuration.posRelative.direction = 0) AND (configuration.posRelative.distance >= 0.0)
                            )(* Sign of distance is evaluated*)
                            OR
                            (configuration.posRelative.direction = FORWARD_DIR)(* Forward direction*)
                            THEN
                            statPosition := ABS(configuration.posRelative.distance);
                           (* Reset MC_MOVERELATIVE command*)
                            instMoveRelative(Axis := axis,
                                             Execute := FALSE);

                            statApplicativeBasicMotionError := FALSE;

                        ELSIF ((configuration.posRelative.direction = 0) AND (configuration.posRelative.distance < 0.0)
                            )(* Sign of distance is evaluated*)
                            OR
                            (configuration.posRelative.direction = BACKWARD_DIR)(* Backward direction*)
                            THEN
                            statPosition := -ABS(configuration.posRelative.distance);
                           (* Reset MC_MOVERELATIVE command*)
                            instMoveRelative(Axis := axis,
                                             Execute := FALSE);

                            statApplicativeBasicMotionError := FALSE;

                        ELSE
                           (* Errorhandling - Invalid direction*)
                            statStatus                      := ERR_INVALID_POS_RELATIVE_DIR;
                            statErrorAutoCleared            := TRUE;
                            diagnostics.subfunctionStatus   := 0;
                            diagnostics                     := statDiagnostics;
                            statApplicativeBasicMotionError := TRUE;
                           (* Set next state*)
                            statFBState          := AXIS_STOP_ON_ERROR_SELECTION;
                            statBasicMotionState := NO_SELECTION;
                        END_IF;
                    END_IF;

                    IF (statApplicativeBasicMotionError = FALSE) THEN
                       (* Call MC_Command*)
                        instMoveRelative(Axis := axis,
                                         Execute := statBasicCommand.5 OR statFirstCycleBasicMotion,(* Input: posRelative*)
                                         Distance := statPosition,
                                         Velocity := configuration.posRelative.velocity,
                                         Acceleration := configuration.posRelative.acceleration,
                                         Deceleration := configuration.posRelative.deceleration,
                                         Jerk := configuration.posRelative.jerk);

                       (* Evaluate MC_Command*)
                        IF (instMoveRelative.Busy = FALSE) AND
                            (instMoveRelative.Error = FALSE) AND
                            (instMoveRelative.Done = FALSE) AND
                            (instMoveRelative.CommandAborted = FALSE)
                            THEN
                           (* Return to NO_SELECTION if command finished*)
                            statBasicMotionState := NO_SELECTION;

                        ELSIF (instMoveRelative.Error = TRUE) THEN
                           (* Errorhandling*)
                            statStatus                    := ERR_MC_MOVERELATIVE;
                            statErrorAutoCleared          := TRUE;
                            diagnostics                   := statDiagnostics;
                            diagnostics.subfunctionStatus := instMoveRelative.ErrorId;
                           (* Set next state*)
                            statFBState          := AXIS_STOP_ON_ERROR_SELECTION;
                            statBasicMotionState := NO_SELECTION;
                        ELSE
                            ;(* Command selected*)
                        END_IF;

                       (* Write MC_Command outputs to internal variable*)
                        statExeOfBasicMotion   := 16#0;
                        statExeOfBasicMotion.0 := instMoveRelative.Busy;
                        statExeOfBasicMotion.1 := instMoveRelative.Done;
                        statExeOfBasicMotion.2 := instMoveRelative.CommandAborted;
                        statExeOfBasicMotion.3 := instMoveRelative.Error;

                    ELSE
                        ;(* Direction not valid*)
                    END_IF;
                {END_REGION}

                POS_ABSOLUTE_SELECTED:
                   (* Additional features (applicative): Change setpoint on the fly (Velocity and Position)*)
                    {REGION "POS_ABSOLUTE_SELECTED"}
                   (* Firstcycle of command*)
                    IF (statFirstCycleBasicMotion = TRUE) THEN
                       (* Reset MC_MOVEABSOLUTE command*)
                        instMoveAbsolute(Axis := axis,
                                         Execute := FALSE);

                        statPosition     := configuration.posAbsolute.position;
                        statVelocity     := configuration.posAbsolute.velocity;    (* Store the last adjusted velocity value*)
                        statAcceleration := configuration.posAbsolute.acceleration;(* Store the last adjusted accerlation value*)
                        statDeceleration := configuration.posAbsolute.deceleration;(* Store the last adjusted deceleration value*)
                        statJerk         := configuration.posAbsolute.jerk;        (* Store the last adjusted jerk value*)
                        statDirection    := configuration.posAbsolute.direction;

                        statVelocityChangeOnTheFly := configuration.posAbsolute.velocityChangeOnTheFly;
                        statPositionChangeOnTheFly := configuration.posAbsolute.positionChangeOnTheFly;

                    ELSIF (((statVelocityChangeOnTheFly = TRUE) AND (configuration.posAbsolute.velocity <> statVelocity)) OR
                        ((statPositionChangeOnTheFly = TRUE) AND (configuration.posAbsolute.position <> statPosition))) AND
                        (instMoveAbsolute.CommandAborted = FALSE)
                        THEN
                        instMoveAbsolute(Axis := axis,
                                         Execute := FALSE);

                        IF (statVelocityChangeOnTheFly = TRUE) THEN(* Apply the new velocity value*)
                            statVelocity := configuration.posAbsolute.velocity;
                        END_IF;

                        IF (statPositionChangeOnTheFly = TRUE) THEN(* Apply the new position value*)
                            statPosition := configuration.posAbsolute.position;
                        END_IF;

                       (* Reset MC_MOVEABSOLUTE command*)
                        instMoveAbsolute(Axis := axis,
                                         Execute := FALSE);
                    END_IF;

                    instMoveAbsolute(Axis := axis,
                                     Execute := statBasicCommand.6 OR statFirstCycleBasicMotion,(* Input: posAbsolute*)
                                     Position := statPosition,
                                     Velocity := statVelocity,
                                     Acceleration := statAcceleration,
                                     Deceleration := statDeceleration,
                                     Jerk := statJerk,
                    (*Direction :=  statDirection*) );

                   (* Evaluate MC_Command*)
                    IF (instMoveAbsolute.Busy = FALSE) AND
                        (instMoveAbsolute.Error = FALSE) AND
                        (instMoveAbsolute.Done = FALSE) AND
                        (instMoveAbsolute.CommandAborted = FALSE)
                        THEN
                       (* Return to NO_SELECTION if command finished*)
                        statBasicMotionState := NO_SELECTION;

                    ELSIF (instMoveAbsolute.Error = TRUE) THEN
                       (* Errorhandling*)
                        statStatus                    := ERR_MC_MOVEABSOLUTE;
                        statErrorAutoCleared          := TRUE;
                        diagnostics                   := statDiagnostics;
                        diagnostics.subfunctionStatus := instMoveAbsolute.ErrorId;
                        statVelocityChangeOnTheFly    := FALSE;
                        statPositionChangeOnTheFly    := FALSE;
                       (* Set next state*)
                        statFBState          := AXIS_STOP_ON_ERROR_SELECTION;
                        statBasicMotionState := NO_SELECTION;

                    ELSE
                        ;(* Command selected*)
                    END_IF;

                   (* Write MC_Command outputs to internal variable*)
                    statExeOfBasicMotion   := 16#0;
                    statExeOfBasicMotion.0 := instMoveAbsolute.Busy;
                    statExeOfBasicMotion.1 := instMoveAbsolute.Done;
                    statExeOfBasicMotion.2 := instMoveAbsolute.CommandAborted;
                    statExeOfBasicMotion.3 := instMoveAbsolute.Error;
                {END_REGION}

                ACTIVE_HOMING_SELECTED:
                   (* Additional fearure (applicative): homing on fixed stop*)
                    {REGION "ACTIVE_HOMING_SELECTED"}
                   (* Firstcycle of command*)
                    IF (statFirstCycleBasicMotion = TRUE) THEN
                        statActiveHomingState  := configuration.homing.extendedMode;
                        statExeOfBasicMotion   := CMD_BUSY;
                        statPassiveHomingState := NO_HOMING_ACTIVE;
                    END_IF;

                   (* Selection of extended homing mode  *)
                    CASE statActiveHomingState OF
                        STANDARD_HOMING:
                           (* No additional features*)
                            {REGION "STANDARD_HOMING"}
                           (* Firstcycle of command*)
                            IF (statFirstCycleBasicMotion = TRUE) THEN
                               (* Reset MC_HOME command*)
                                instHome(Axis := axis,
                                         bCalibrationCam := homingSensor,
                                         Execute := FALSE);

                               (* Reset TON command*)
                                instTimerTON(IN := FALSE,
                                             PT := configuration.homing.homeExecutionTimeLimit);
                            END_IF;

                           (* Call MC_Command*)
                            instHome(Axis := axis,
                                     bCalibrationCam := homingSensor,
                                     Execute := statBasicCommand.10 OR statFirstCycleBasicMotion,(* Input: homing*)
                                     Position := configuration.homing.position,
                            (*Mode :=  configuration.homing.mode*) );

                           (*Call TON*)
                            instTimerTON(IN := TRUE,
                                         PT := configuration.homing.homeExecutionTimeLimit);

                           (* Evaluate MC_Command*)
                            IF (instHome.Busy = FALSE) AND
                                (instHome.Done = FALSE) AND
                                (instHome.CommandAborted = FALSE) AND
                                (instHome.Error = FALSE)
                                THEN
                               (* Return to NO_SELECTION if command finished*)
                                statActiveHomingState := STANDARD_HOMING;
                                statBasicMotionState  := NO_SELECTION;

                            ELSIF (instHome.Error = TRUE OR instTimerTON.Q) THEN
                               (* Errorhandling*)
                                statStatus                    := ERR_MC_HOME;
                                statErrorAutoCleared          := TRUE;
                                diagnostics                   := statDiagnostics;
                                diagnostics.subfunctionStatus := instHome.ErrorId;
                                statFBState                   := AXIS_STOP_ON_ERROR_SELECTION;
                                statBasicMotionState          := NO_SELECTION;

                            ELSE
                                ;(* Command selected*)

                            END_IF;

                            statExeOfBasicMotion   := 16#0;
                            statExeOfBasicMotion.0 := instHome.Busy;
                            statExeOfBasicMotion.1 := instHome.Done;
                            statExeOfBasicMotion.2 := instHome.CommandAborted;
                            statExeOfBasicMotion.3 := instHome.Error;
                        {END_REGION}
                        HOMING_ON_FIXED_STOP:
                           (* This case is additional feature (MC_MOVEVELOCITY and MC_HOME internal used)*)
                            {REGION "REFERENCE_TO_FIXED_STOP"}
                            CASE statExeOfBasicMotion OF
                                CMD_BUSY:
                                   (* Firstcycle of command*)
                                    IF (statFirstCycleBasicMotion = TRUE) THEN
                                       (* Check if homing on fixed stop is allowed  *)
                                        (*IF ( axis.Modulo.Enable = TRUE) THEN*)
                                        IF (tempFalse = TRUE) THEN
                                           (* Modulo enabled - Errorhandling*)
                                            statStatus                    := ERR_MODULO_NOT_ALLOWED;
                                            statErrorAutoCleared          := TRUE;
                                            diagnostics.subfunctionStatus := 0;
                                            diagnostics.basicMotionState  := statBasicMotionState;
                                           (* Set next state*)
                                            statFBState           := AXIS_STOP_ON_ERROR_SELECTION;
                                            statBasicMotionState  := NO_SELECTION;
                                            statActiveHomingState := STANDARD_HOMING;
                                            statHomingSubState    := HOMING_IDLE;

                                        ELSIF (configuration.homing.extendedModeTorqueLimit = 0)(* Torqueliming 0 in configuration *)
                                            THEN
                                           (* Errorhandling -  Torquevalue 0 configured*)
                                            statStatus                    := ERR_INVALID_TORQUE_LIMIT;
                                            statErrorAutoCleared          := TRUE;
                                            diagnostics.subfunctionStatus := 0;
                                            diagnostics.basicMotionState  := statBasicMotionState;
                                           (* Set next state*)
                                            statFBState           := AXIS_STOP_ON_ERROR_SELECTION;
                                            statBasicMotionState  := NO_SELECTION;
                                            statActiveHomingState := STANDARD_HOMING;
                                            statHomingSubState    := HOMING_IDLE;

                                            (*ELSIF ( axis.Homing.ReferencingVelocity = 0)*)
                                        ELSIF (configuration.homing.offsetPositionVelocity = 0)
                                            THEN
                                           (* Errorhandling -  Velocity 0 configured*)
                                            statStatus                    := ERR_INVALID_VELOCITY;
                                            statErrorAutoCleared          := TRUE;
                                            diagnostics.subfunctionStatus := 0;
                                            diagnostics.basicMotionState  := statBasicMotionState;
                                           (* Set next state*)
                                            statFBState           := AXIS_STOP_ON_ERROR_SELECTION;
                                            statBasicMotionState  := NO_SELECTION;
                                            statActiveHomingState := STANDARD_HOMING;
                                            statHomingSubState    := HOMING_IDLE;

                                        ELSE
                                           (* Store dynamic values*)
                                            (*statHomingPosition :=  configuration.homing.position;
	                             statVelocity :=  axis.Homing.ReferencingVelocity;
	                             statAcceleration :=  axis.DynamicDefaults.Acceleration;
	                             statDeceleration :=  axis.DynamicDefaults.Deceleration;
	                             statJerk :=  axis.DynamicDefaults.Jerk;
	                             statTorqueLimit :=  configuration.homing.extendedModeTorqueLimit;*)
                                            statHomingPosition := configuration.homing.position;
                                            statVelocity       := configuration.homing.offsetPositionVelocity;
                                            statAcceleration   := configuration.homing.offsetPositionAcceleration;
                                            statDeceleration   := configuration.homing.offsetPositonDeceleration;
                                            statJerk           := configuration.homing.offsetPositionJerk;
                                            statTorqueLimit    := configuration.homing.extendedModeTorqueLimit;

                                           (* Detecting operating sensor*)
                                            (*
								FOR  tempIndex := 1 TO 4 DO
	                              IF  axis.StatusSensor[ tempIndex].Control = TRUE
	                              THEN
	                                EXIT;
	                              END_IF;
	                            END_FOR;
	                            *)
                                            (*IF ( axis.Sensor[ tempIndex].ActiveHoming.Direction = 0)(* Positve direction configured*)
	                            THEN*)
                                           (* Positive direction*)
                                            statDirection := FORWARD_DIR;
                                            (* ELSE
	                             (* Negative direction*)
	                               statDirection :=  BACKWARD_DIR;
	                            END_IF;
	                            *)
                                            (*statTorqueLimitingState :=  FIXED_STOP_DETECTION_ACTIVE;*)
                                           (* Reset MC_Commands*)
                                            instHome(Axis := axis,
                                                     bCalibrationCam := homingSensor,
                                                     Execute := FALSE);

                                            instMoveVelocity(Axis := axis,
                                                             Execute := FALSE);

                                            instMoveAbsolute(Axis := axis,
                                                             Execute := FALSE);

                                           (* Reset TON*)
                                            instTimerTON(IN := FALSE,
                                                         PT := configuration.homing.homeExecutionTimeLimit);

                                           (* Determine the encoder type*)
                                            (* tempIndex := 1;
	                             tempIndex := UDINT_TO_INT( axis.OperativeSensor);
	                            IF ( axis.Sensor[ tempIndex].Type =  INCREMENTAL_ENCODER) THEN
	                               statHomingMode :=  DIRECT_HOMING; // Direct homing (absolute)
	                            ELSE
	                               statHomingMode :=  ABSOLUTE_ENCODER_ADJUSTMENT;
	                            END_IF;
								*)
                                           (* Use always direct homing*)
                                           (* statHomingMode :=  DIRECT_HOMING; // Direct homing (absolute)*)
                                           (* Set next state*)
                                            (*statHomingSubState :=  HOMING_FIXED_STOP_DETECTION;*)
                                            statHomingSubState := HOMING_PROCESS;
                                        END_IF;
                                    END_IF;

                                   (* Call OF subStateMachine*)
                                    REPEAT
                                        CASE statHomingSubState OF
                                            HOMING_IDLE:
                                                tempStateChangeActive := FALSE;
                                                ;(* Do nothing, inserted no exectution of homing if error occurred in first cycle*)

                                            HOMING_FIXED_STOP_DETECTION:
                                                tempStateChangeActive := FALSE;

                                               (* Start axis to detect fixed stop*)
                                                instMoveVelocity(Axis := axis,
                                                                 Execute := TRUE,
                                                                 Velocity := statVelocity,
                                                                 Acceleration := statAcceleration,
                                                                 Deceleration := statDeceleration,
                                                                 Jerk := statJerk,
                                                (*PositionControlled := TRUE,*)
                                                (*Direction :=  statDirection*) );

                                               (* Read Statusword only when not already read out*)
                                                IF (tempStatusWord = 16#0)
                                                    THEN
                                                    (*tempStatusWord :=  axis.StatusWord;*)
                                                    tempStatusWord := axis.NcToPlc.StateDWord;
                                                END_IF;

                                               (* Evaluate MC_Command*)
                                                IF (tempStatusWord.30 = TRUE) THEN(* inClamping = TRUE*)
                                                   (* Fixed stop detected --> start homing process*)
                                                    statHomingSubState    := HOMING_PROCESS;
                                                    tempStateChangeActive := TRUE;

                                                ELSIF (instMoveVelocity.Error = TRUE) THEN
                                                   (* Errorhandling*)
                                                    statStatus                    := ERR_MC_MOVEVELOCITY;
                                                    statErrorAutoCleared          := TRUE;
                                                    diagnostics                   := statDiagnostics;
                                                    diagnostics.subfunctionStatus := instMoveVelocity.ErrorId;
                                                   (* Set next state*)
                                                    statFBState           := AXIS_STOP_ON_ERROR_SELECTION;
                                                    statBasicMotionState  := NO_SELECTION;
                                                    statActiveHomingState := STANDARD_HOMING;
                                                    statExeOfBasicMotion  := CMD_ERROR;
                                                    statHomingSubState    := HOMING_IDLE;

                                                ELSIF (instMoveVelocity.CommandAborted = TRUE) THEN
                                                   (* Set next state*)
                                                    statExeOfBasicMotion := CMD_ABORTED;
                                                    statHomingSubState   := HOMING_IDLE;

                                                ELSE
                                                    ;(* Wait for detecting fixed stop*)
                                                END_IF;

                                            HOMING_PROCESS:
                                                tempStateChangeActive := FALSE;
                                               (* Execute MC_HOME*)
                                                instHome(Axis := axis,
                                                         bCalibrationCam := homingSensor,
                                                         Execute := TRUE,
                                                         Position := statHomingPosition,
                                                (*Mode :=  statHomingMode*) );

                                               (*Call TON*)
                                                instTimerTON(IN := TRUE,
                                                             PT := configuration.homing.homeExecutionTimeLimit);

                                               (* Evaluate MC_Command*)
                                                IF (instHome.Done = TRUE) THEN
                                                   (* MC_HOME finished - Set next state*)
                                                    statHomingSubState    := HOMING_POSITION;
                                                    tempStateChangeActive := TRUE;
                                                    instTimerTON.IN       := FALSE;

                                                ELSIF (instHome.Error = TRUE OR instTimerTON.Q) THEN
                                                   (* Errorhandling*)
                                                    statStatus                    := ERR_MC_HOME;
                                                    statErrorAutoCleared          := TRUE;
                                                    diagnostics                   := statDiagnostics;
                                                    diagnostics.subfunctionStatus := instHome.ErrorId;
                                                   (* Set next state*)
                                                    statFBState          := AXIS_STOP_ON_ERROR_SELECTION;
                                                    statExeOfBasicMotion := CMD_ERROR;
                                                    statHomingSubState   := HOMING_IDLE;

                                                ELSIF (instHome.CommandAborted = TRUE) THEN
                                                   (* Set next state*)
                                                    statExeOfBasicMotion := CMD_ABORTED;
                                                    statHomingSubState   := HOMING_IDLE;
                                                ELSE
                                                    ;(* Wait for finish homing process*)
                                                END_IF;

                                            HOMING_POSITION:
                                                tempStateChangeActive := FALSE;

                                                statHomingPosition := configuration.homing.offsetPosition;
                                                statVelocity       := configuration.homing.offsetPositionVelocity;
                                                statAcceleration   := configuration.homing.offsetPositionAcceleration;
                                                statDeceleration   := configuration.homing.offsetPositonDeceleration;
                                                statJerk           := configuration.homing.offsetPositionJerk;

                                               (* Execute moving to homeposition*)
                                                instMoveAbsolute(Axis := axis,
                                                                 Execute := TRUE,
                                                                 (*Position :=  statHomingPosition,*)
                                                                 Position := configuration.homing.offsetPosition,
                                                                 Velocity := ABS(statVelocity),
                                                                 Acceleration := statAcceleration,
                                                                 Deceleration := statDeceleration,
                                                                 Jerk := statJerk,
                                                (*Direction :=  SHORTEST_WAY_DIR*) );

                                               (* Evaluate MC_Command*)
                                                IF (instMoveAbsolute.Done = TRUE) THEN
                                                   (* Homeposition reached - Set next state*)
                                                    statExeOfBasicMotion := CMD_DONE;
                                                    statHomingSubState   := HOMING_IDLE;

                                                ELSIF (instMoveAbsolute.Error = TRUE) THEN
                                                   (* Errorhandling*)
                                                    statStatus                    := ERR_MC_MOVEABSOLUTE;
                                                    statErrorAutoCleared          := TRUE;
                                                    diagnostics                   := statDiagnostics;
                                                    diagnostics.subfunctionStatus := instMoveAbsolute.ErrorId;
                                                   (* Set next state*)
                                                    statFBState           := AXIS_STOP_ON_ERROR_SELECTION;
                                                    statBasicMotionState  := CMD_BUSY;
                                                    statActiveHomingState := STANDARD_HOMING;
                                                    statExeOfBasicMotion  := CMD_ERROR;
                                                    statHomingSubState    := HOMING_IDLE;

                                                ELSIF (instMoveAbsolute.CommandAborted = TRUE) THEN
                                                   (* Set next state*)
                                                    statExeOfBasicMotion := CMD_ABORTED;
                                                    statHomingSubState   := HOMING_IDLE;

                                                ELSE
                                                    ;(* Wait for reaching homeposition*)
                                                END_IF;

                                        ELSE
                                           (* Errorhandling *)
                                            statStatus                    := ERR_UNDEFINED_EXTENDED_HOMING_SUBSTATE;
                                            statErrorUserCleared          := TRUE;
                                            diagnostics                   := statDiagnostics;
                                            diagnostics.subfunctionStatus := 0;
                                           (* Set errorstate*)
                                            statFBState           := FB_ERROR;
                                            tempStateChangeActive := FALSE;
                                        END_CASE;

                                    UNTIL (tempStateChangeActive = FALSE)(* Repeat execution if a state is changing*)
                                    END_REPEAT;

                                CMD_DONE,
                                    CMD_ABORTED,
                                    CMD_ERROR:
                                   (* Return to NO_SELECTION if command finished*)
                                    IF (statBasicCommand.10 = FALSE)(* homing = FALSE*)
                                        THEN
                                       (* Return to NO_HOMING_ACTIVE if command finished*)
                                        statBasicMotionState  := NO_SELECTION;
                                        statActiveHomingState := STANDARD_HOMING;
                                        statExeOfBasicMotion  := CMD_BUSY;
                                        statHomingSubState    := HOMING_IDLE;
                                    ELSE
                                        ;(* Wait for falling edge at homing command*)
                                    END_IF;

                            ELSE
                               (* Errorhandling*)
                                statStatus                    := ERR_UNDEFINED_EXTENDED_HOMING_STATE;
                                statErrorUserCleared          := TRUE;
                                diagnostics                   := statDiagnostics;
                                diagnostics.subfunctionStatus := 0;
                               (* Set errorstate*)
                                statFBState := FB_ERROR;
                            END_CASE;
                    {END_REGION}

                    ELSE
                       (* Errorhandling*)
                        statStatus                    := ERR_INVALID_HOMING_EXTENDED_MODE;
                        statErrorAutoCleared          := TRUE;
                        diagnostics                   := statDiagnostics;
                        diagnostics.subfunctionStatus := 0;
                       (* Set next state*)
                        statFBState           := AXIS_STOP_ON_ERROR_SELECTION;
                        statBasicMotionState  := NO_SELECTION;
                        statActiveHomingState := STANDARD_HOMING;
                        statBasicMotionState  := NO_SELECTION;
                    END_CASE;
                {END_REGION}

                GEAR_IN_RELATIVE_SELECTED:
                   (* Additional features (applicative): Change setpoint on the fly (gear ratio)*)
                    {REGION "GEAR_IN_RELATIVE_SELECTED"}
                   (* Firstcycle of command*)
                    IF (statFirstCycleBasicMotion = TRUE) THEN
                       (* Reset GEAR_IN command *)
                        instGearIn(Master := master,
                                   Slave := axis,
                                   Execute := FALSE);

                        (*statRatioNumerator :=  configuration.gearInRelative.ratioNumerator;*)
                        statRatioNumerator      := configuration.gearInRelative.ratioDenominator;
                        statRatioDenominator    := configuration.gearInRelative.ratioDenominator;
                        statAcceleration        := configuration.gearInRelative.acceleration;
                        statDeceleration        := configuration.gearInRelative.deceleration;
                        statJerk                := configuration.gearInRelative.jerk;
                        statRatioChangeOnTheFly := configuration.gearInRelative.ratioChangeOnTheFly;

                    ELSIF ((statRatioChangeOnTheFly = TRUE)(* Flying change of ratio numerator*)
                    (*AND (( configuration.gearInRelative.ratioNumerator <>  statRatioNumerator)*)
                        AND
                        ((configuration.gearInRelative.ratioDenominator <> statRatioNumerator) OR
                        (configuration.gearInRelative.ratioDenominator <> statRatioDenominator))) AND
                        (instGearIn.CommandAborted = FALSE)
                        THEN
                        instGearIn(Master := master,
                                   Slave := axis,
                                   Execute := FALSE);

                        statRatioNumerator   := configuration.gearInRelative.ratioDenominator;(* Apply the new gear ratio numerator*)
                        statRatioDenominator := configuration.gearInRelative.ratioDenominator;(* Apply the new gear ratio denominator*)
                    END_IF;

                   (* Call MC_Command*)
                    instGearIn(Master := master,
                               Slave := axis,
                               Execute := statBasicCommand.7 OR statFirstCycleBasicMotion,(* Input: gearInRelative*)
                               RatioNumerator := statRatioNumerator,
                               RatioDenominator := DINT_TO_UINT(statRatioDenominator),
                               Acceleration := statAcceleration,
                               Deceleration := statDeceleration,
                               Jerk := statJerk);

                   (* Evaluate MC_Command*)
                    IF (instGearIn.Busy = FALSE) AND
                        (instGearIn.Error = FALSE) AND
                        (instGearIn.CommandAborted = FALSE) AND
                        (instGearIn.InGear = FALSE)
                        THEN
                       (* Return to NO_SELECTION if command finished*)
                        statBasicMotionState := NO_SELECTION;

                    ELSIF (instGearIn.Error = TRUE) THEN
                       (* Errorhandling*)
                        statStatus                    := ERR_MC_GEARIN;
                        statErrorAutoCleared          := TRUE;
                        diagnostics                   := statDiagnostics;
                        diagnostics.subfunctionStatus := instGearIn.ErrorId;
                        statRatioChangeOnTheFly       := FALSE;
                       (* Set next state*)
                        statFBState          := AXIS_STOP_ON_ERROR_SELECTION;
                        statBasicMotionState := NO_SELECTION;

                    ELSE
                        ;(* Command selected*)
                    END_IF;

                   (* Read Statusword only when not already read out*)
                    IF ( tempStatusWord = 16#0)
                    THEN

                       tempStatusWord :=  axis.NcToPlc.StateDWord;

                    END_IF;

                   (* Write MC_Command outputs to internal variable*)
                    statExeOfBasicMotion   := 16#0;
                    statExeOfBasicMotion.0 := instGearIn.Busy;
                    statExeOfBasicMotion.2 := instGearIn.CommandAborted;
                    statExeOfBasicMotion.3 := instGearIn.Error;
                   (* statExeOfBasicMotion.6 :=  tempStatusWord.21 AND NOT  instGearIn.InGear; // write Synchronizing only when bit of instance of MC_GearIn.InGear = FALSE*)
                    statExeOfBasicMotion.7 := instGearIn.InGear;
                {END_REGION}

                GEAR_IN_ABSOLUTE_SELECTED:
                   (* Additional features (applicative): Change setpoint on the fly (gear ratio)*)
                    {REGION "GEAR_IN_SELECTED"}
                   (* Firstcycle of command*)
                    IF (statFirstCycleBasicMotion = TRUE) THEN
                       (* Reset GEAR_IN_POS command *)
                        instGearInPos(Master := master,
                                      Slave := axis,
                        (*Execute := FALSE*) );

                        statRatioNumerator       := configuration.gearInAbsolute.ratioNumerator;
                        statRatioDenominator     := configuration.gearInAbsolute.ratioDenominator;
                        statMasterSyncPosition   := configuration.gearInAbsolute.masterSyncPosition;
                        statSlaveSyncPosition    := configuration.gearInAbsolute.slaveSyncPosition;
                        statSyncProfileReference := configuration.gearInAbsolute.syncProfileReference;
                        statMasterStartDistance  := configuration.gearInAbsolute.masterStartDistance;
                        statVelocity             := configuration.gearInAbsolute.velocity;
                        statAcceleration         := configuration.gearInAbsolute.acceleration;
                        statDeceleration         := configuration.gearInAbsolute.deceleration;
                        statJerk                 := configuration.gearInAbsolute.jerk;
                        statSyncDirection        := configuration.gearInAbsolute.syncDirection;
                        statRatioChangeOnTheFly  := configuration.gearInAbsolute.ratioChangeOnTheFly;

                    ELSIF (((statRatioChangeOnTheFly = TRUE) AND (configuration.gearInAbsolute.ratioNumerator <> statRatioNumerator)) OR
                        ((statRatioChangeOnTheFly = TRUE) AND (configuration.gearInAbsolute.ratioDenominator <> statRatioDenominator))) AND
                        (instGearInPos.CommandAborted = FALSE)
                        THEN
                        instGearInPos(Master := master,
                                      Slave := axis,
                        			Enable := FALSE );

                        statRatioNumerator   := configuration.gearInAbsolute.ratioNumerator;  (* Apply the new gear ratio numerator*)
                        statRatioDenominator := configuration.gearInAbsolute.ratioDenominator;(* Apply the new gear ratio denominator*)
                    END_IF;

